(* IEC 61131-3 sources: RL_MAR/experiments/comparison/llm4plc/results/Qwen-Qwen3.5-9B_20260506_150728/20260506_164922, 2 files *)

(* ---- generated_code_iteration_0.st ---- *)
START_ST
FUNCTION_BLOCK WindTurbineControl
VAR_INPUT
    WindSpeedSensor : REAL; (* Input for measuring wind speed *)
    GeneratorSpeedSensor : REAL; (* Input for measuring generator speed *)
END_VAR

VAR_OUTPUT
    BladePitch : INT; (* Output for blade pitch control (degrees) *)
    GeneratorSpeed : REAL; (* Output for generator speed control (RPM) *)
END_VAR

VAR
    currentWindState : INT; // THE STATE VARIABLE TRACKING CURRENT WIND CONDITION
    targetBladePitch : INT; // INTERMEDIATE VARIABLE TO HOLD CALCULATED PITCH
    targetGenSpeed : REAL; // INTERMEDIATE VARIABLE TO HOLD CALCULATED SPEED
    windSpeedSensor : REAL; // INPUT VARIABLE (SHADOW COPY FOR LOGIC CLARITY)
    generatorSpeedSensor : REAL; // INPUT VARIABLE (SHADOW COPY FOR LOGIC CLARITY)
END_VAR

(* Initialize state to LOW_WIND_MODE (0) on first execution or reset *)
IF currentWindState = 0 AND (NOT (WindSpeedSensor > 3.0)) THEN
    currentWindState := 0;
ELSIF currentWindState = 0 AND (WindSpeedSensor > 3.0) THEN
    currentWindState := 1;
ELSIF currentWindState = 1 AND (WindSpeedSensor <= 3.0) THEN
    currentWindState := 0;
ELSIF currentWindState = 1 AND (WindSpeedSensor > 5.0) THEN
    currentWindState := 2;
ELSIF currentWindState = 2 AND (WindSpeedSensor <= 5.0) THEN
    currentWindState := 1;
ELSIF currentWindState = 2 AND (WindSpeedSensor <= 3.0) THEN
    currentWindState := 0; (* Direct jump to lowest state if wind drops significantly *)
END_IF

(* Assign output values based on the determined state *)
CASE currentWindState OF
    0: (* LOW_WIND_MODE *)
        targetBladePitch := -5;
        targetGenSpeed := 500.0;
    1: (* MODERATE_WIND_MODE *)
        targetBladePitch := 0;
        targetGenSpeed := 800.0;
    2: (* HIGH_WIND_MODE *)
        targetBladePitch := 5;
        targetGenSpeed := 1000.0;
END_CASE

(* Assign calculated targets to actual outputs *)
BladePitch := targetBladePitch;
GeneratorSpeed := targetGenSpeed;

END_FUNCTION_BLOCK
END_ST

(* ---- generated_code_iteration_1.st ---- *)
START_REASON
The validation feedback indicates a variable shadowing error in the CODESYS compiler. Specifically, the local variable `windSpeedSensor` (and `generatorSpeedSensor`) is defined in the `VAR` section, but it has the exact same name as the input variables `WindSpeedSensor` and `GeneratorSpeedSensor` defined in the `VAR_INPUT` section. In IEC 61131-3 Structured Text, local variables cannot have the same name as inputs or outputs of the same function block, as this causes ambiguity and compilation errors.

To fix this:
1.  Remove the redundant local variables `windSpeedSensor` and `generatorSpeedSensor` from the `VAR` section.
2.  Update the logic to directly reference the `VAR_INPUT` variables (`WindSpeedSensor` and `GeneratorSpeedSensor`) instead of the shadowed local copies.
3.  Ensure the state machine logic remains intact while using the correct input names.
END_REASON

START_ST
FUNCTION_BLOCK WindTurbineControl
VAR_INPUT
    WindSpeedSensor : REAL; (* Input for measuring wind speed *)
    GeneratorSpeedSensor : REAL; (* Input for measuring generator speed *)
END_VAR

VAR_OUTPUT
    BladePitch : INT; (* Output for blade pitch control (degrees) *)
    GeneratorSpeed : REAL; (* Output for generator speed control (RPM) *)
END_VAR

VAR
    currentWindState : INT; // THE STATE VARIABLE TRACKING CURRENT WIND CONDITION
    targetBladePitch : INT; // INTERMEDIATE VARIABLE TO HOLD CALCULATED PITCH
    targetGenSpeed : REAL; // INTERMEDIATE VARIABLE TO HOLD CALCULATED SPEED
END_VAR

(* Initialize state to LOW_WIND_MODE (0) on first execution or reset *)
IF currentWindState = 0 AND (NOT (WindSpeedSensor > 3.0)) THEN
    currentWindState := 0;
ELSIF currentWindState = 0 AND (WindSpeedSensor > 3.0) THEN
    currentWindState := 1;
ELSIF currentWindState = 1 AND (WindSpeedSensor <= 3.0) THEN
    currentWindState := 0;
ELSIF currentWindState = 1 AND (WindSpeedSensor > 5.0) THEN
    currentWindState := 2;
ELSIF currentWindState = 2 AND (WindSpeedSensor <= 5.0) THEN
    currentWindState := 1;
ELSIF currentWindState = 2 AND (WindSpeedSensor <= 3.0) THEN
    currentWindState := 0; (* Direct jump to lowest state if wind drops significantly *)
END_IF

(* Assign output values based on the determined state *)
CASE currentWindState OF
    0: (* LOW_WIND_MODE *)
        targetBladePitch := -5;
        targetGenSpeed := 500.0;
    1: (* MODERATE_WIND_MODE *)
        targetBladePitch := 0;
        targetGenSpeed := 800.0;
    2: (* HIGH_WIND_MODE *)
        targetBladePitch := 5;
        targetGenSpeed := 1000.0;
END_CASE

(* Assign calculated targets to actual outputs *)
BladePitch := targetBladePitch;
GeneratorSpeed := targetGenSpeed;

END_FUNCTION_BLOCK
END_ST
